Yaskawa INFORM job: pipe_head_cone_program.JBI

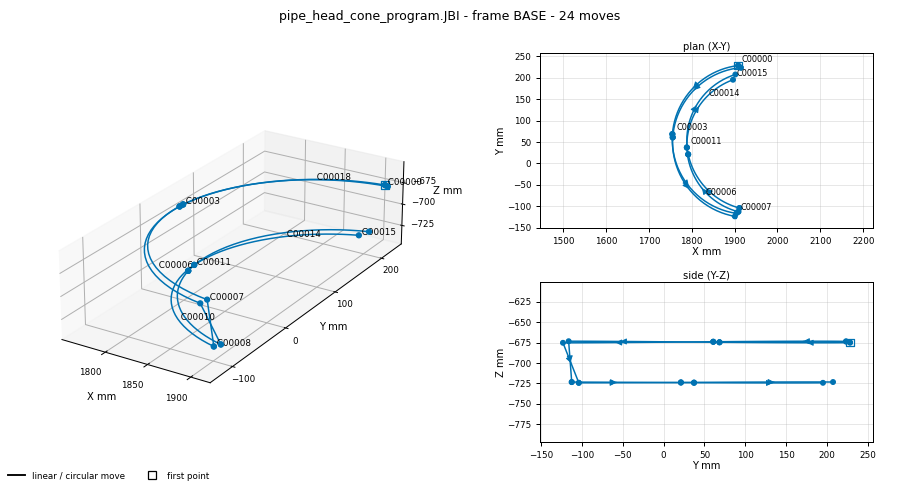
[picture p0: tool path of pipe_head_cone_program.JBI in frame BASE, 24 of 36 moves have a stored position in this frame; points joined in program order, loops and branches not executed]
/JOB
//NAME pipe_head_cone_program
//POS
///NPOS 32,0,32,0,0,0
///TOOL 0
///POSTYPE BASE
///RECTAN
///RCONF 0,0,0,0,0,0,0,0,0,0,0,0,0,0,0,0,0,0,0,0,0,0,0,0
C00000=1908.636152,228.405172,-674.878909,180.000000,-60.000000,-69.549462
C00001=1908.636152,228.405172,-674.878909,180.000000,-60.000000,-69.549462
C00002=1876.167519,221.329617,-675.039561,180.000000,-60.000000,-59.849757
C00003=1755.071902,68.421903,-674.544265,180.000000,-60.000000,-4.153835
C00004=1755.071902,68.421903,-674.544265,180.000000,-60.000000,-4.153835
C00005=1755.071902,68.421903,-674.544265,180.000000,-60.000000,-4.153835
C00006=1822.450269,-81.635382,-673.353049,180.000000,-60.000000,41.469946
C00007=1904.071832,-116.428639,-673.267963,180.000000,-60.000000,67.447139
C00008=1908.955628,-112.668557,-723.335713,180.000000,-60.000000,68.184011
C00009=1908.955628,-112.668557,-723.335713,180.000000,-60.000000,68.184011
C00010=1847.316751,-81.398855,-723.439739,180.000000,-60.000000,46.193571
C00011=1788.752080,37.201124,-724.061997,180.000000,-60.000000,4.334492
C00012=1788.752080,37.201124,-724.061997,180.000000,-60.000000,4.334492
C00013=1788.752080,37.201124,-724.061997,180.000000,-60.000000,4.334492
C00014=1829.773030,149.694365,-724.362002,180.000000,-60.000000,-34.198094
C00015=1896.448255,195.225334,-724.211350,-180.000000,-60.000000,-61.504475
C00016=1914.567024,223.493965,-673.539997,-180.000000,-60.000000,-70.848369
C00017=1914.567024,223.493965,-673.539997,-180.000000,-60.000000,-70.848369
C00018=1838.192764,197.573782,-673.255407,180.000000,-60.000000,-47.506196
C00019=1755.800316,60.783986,-673.903618,180.000000,-60.000000,-3.460700
C00020=1755.800316,60.783986,-673.903618,180.000000,-60.000000,-3.460700
C00021=1755.800316,60.783986,-673.903618,180.000000,-60.000000,-3.460700
C00022=1832.773847,-95.800228,-675.136710,-180.000000,-60.000000,45.073545
C00023=1900.765726,-123.399110,-675.193023,180.000000,-60.000000,66.324251
C00024=1911.422097,-103.974544,-724.211216,180.000000,-60.000000,67.272130
C00025=1911.422097,-103.974544,-724.211216,180.000000,-60.000000,67.272130
C00026=1858.919147,-79.590504,-724.220331,180.000000,-60.000000,47.768783
C00027=1791.910994,21.149631,-723.799652,180.000000,-60.000000,8.540897
C00028=1791.910994,21.149631,-723.799652,180.000000,-60.000000,8.540897
C00029=1791.910994,21.149631,-723.799652,180.000000,-60.000000,8.540897
C00030=1889.422656,203.042247,-723.239264,180.000000,-60.000000,-60.886256
C00031=1901.992103,207.564393,-723.270249,180.000000,-60.000000,-65.206256
///POSTYPE PULSE
///PULSE
EX00000=336896.0
///POSTYPE PULSE
///PULSE
EC00000=153600.0
EC00001=153600.0
EC00002=153600.0
EC00003=153600.0
EC00004=153600.0
EC00005=153600.0
EC00006=153600.0
EC00007=153600.0
EC00008=153600.0
EC00009=153600.0
EC00010=153600.0
EC00011=153600.0
EC00012=153600.0
EC00013=153600.0
EC00014=153600.0
EC00015=153600.0
EC00016=336896.0
EC00017=336896.0
EC00018=336896.0
EC00019=336896.0
EC00020=336896.0
EC00021=336896.0
EC00022=336896.0
EC00023=336896.0
EC00024=336896.0
EC00025=336896.0
EC00026=336896.0
EC00027=336896.0
EC00028=336896.0
EC00029=336896.0
EC00030=336896.0
EC00031=336896.0
//INST
///DATE 2023/08/13 11:14
///ATTR SC,RW,RJ
////FRAME BASE
///GROUP1 RB1,ST1
NOP
MOVJ P009 EX000 VJ=15.00
MOVJ C00000 EC00000 VJ=15.0
CALL JOB:SPYON
MOVC C00001 EC00001 V=150.0
MOVC C00002 EC00002 V=150.0
MOVC C00003 EC00003 V=150.0
MOVL C00004 EC00004 V=150.0
MOVC C00005 EC00005 V=150.0
MOVC C00006 EC00006 V=150.0
MOVC C00007 EC00007 V=150.0
MOVL C00008 EC00008 V=150.0
MOVC C00009 EC00009 V=150.0
MOVC C00010 EC00010 V=150.0
MOVC C00011 EC00011 V=150.0
MOVL C00012 EC00012 V=150.0
MOVC C00013 EC00013 V=150.0
MOVC C00014 EC00014 V=150.0
MOVC C00015 EC00015 V=150.0
CALL JOB:SPYOF
MOVJ P009 VJ=15.00
MOVJ C00016 EC00016 VJ=15.0
CALL JOB:SPYON
MOVC C00017 EC00017 V=150.0
MOVC C00018 EC00018 V=150.0
MOVC C00019 EC00019 V=150.0
MOVL C00020 EC00020 V=150.0
MOVC C00021 EC00021 V=150.0
MOVC C00022 EC00022 V=150.0
MOVC C00023 EC00023 V=150.0
MOVL C00024 EC00024 V=150.0
MOVC C00025 EC00025 V=150.0
MOVC C00026 EC00026 V=150.0
MOVC C00027 EC00027 V=150.0
MOVL C00028 EC00028 V=150.0
MOVC C00029 EC00029 V=150.0
MOVC C00030 EC00030 V=150.0
MOVC C00031 EC00031 V=150.0
CALL JOB:SPYOF
MOVJ P009 VJ=15.00
MOVL P009 EX00000 V=150.0
END
